// TwinCAT 3 PLC project Execution_Options
// ProgramVersion: 3.1.4023.0
// libraries:
//   Tc2_MC2, * (Beckhoff Automation GmbH)
//   Tc2_Standard, * (Beckhoff Automation GmbH)
//   Tc2_System, * (Beckhoff Automation GmbH)
//   Tc3_Module, * (Beckhoff Automation GmbH)
// project tree:
//   Body Execution/ Body_Task_Base.TcPOU, AxesReset_Body.TcPOU
//   Cycle Method/ AxesReset_Cycle.TcPOU, Cyclic_Task_Base.TcPOU
//   / PlcTask.TcTTO
//   POUs/ MAIN.TcPOU
// real-time tasks:
//   TASK PlcTask: cycle T#10ms, priority 20, ADS port 350

CONFIGURATION Execution_Options
    RESOURCE PLC ON TwinCAT3
        TASK PlcTask(INTERVAL := T#10ms, PRIORITY := 20);
        PROGRAM MAIN WITH PlcTask : MAIN;
    END_RESOURCE
END_CONFIGURATION

// ---- POUs/MAIN.TcPOU
PROGRAM MAIN
VAR
	Axis : AXIS_REF;
	BodyExecution_AxisReset : AxesReset_Body(Axis);
	CycleExecution_AxesReset : AxesReset_Cycle(Axis);
	
END_VAR

///////////////Cycle Call for Body execution//////////////
BodyExecution_AxisReset();


///////////////Cycle Call for Cycle execution////////////
CycleExecution_AxesReset.Cycle();

END_PROGRAM

// ---- Body Execution/AxesReset_Body.TcPOU
FUNCTION_BLOCK AxesReset_Body EXTENDS Body_Task_Base
VAR_INPUT
END_VAR
VAR_OUTPUT
END_VAR
VAR
	resetMover : Tc2_MC2.MC_Reset;
	_axis : REFERENCE TO Tc2_MC2.AXIS_REF;
	_ResetMover : BOOL;
	state : INT;

END_VAR

CASE State OF
	0:
		IF _ResetMover THEN
			_done := FALSE;
			_error := FALSE;
			_busy := TRUE;
			resetMover.Execute := TRUE;
			IF resetMover.Busy THEN
				State := 10;
				_ResetMover := FALSE;
			END_IF
		END_IF
	
	10:
		IF NOT resetMover.Busy THEN
			IF resetMover.Done THEN
				_done := TRUE;
			ELSIF resetMover.Error THEN
				_error := TRUE;
			END_IF
			_busy := FALSE;
			resetMover.Execute := FALSE;
			State := 0;
		END_IF
END_CASE

resetMover(Axis := _axis);

METHOD Abort : BOOL
resetMover.Execute := FALSE;
_busy := FALSE;
_ResetMover := FALSE;
Abort := TRUE;
State := 0;
END_METHOD

PROPERTY Busy : BOOL
GET
Busy := _busy;
END_GET
END_PROPERTY

PROPERTY Done : BOOL
GET
Done := _done;
END_GET
END_PROPERTY

PROPERTY Error : BOOL
GET
Error := _error;
END_GET
END_PROPERTY

METHOD Execute : BOOL
VAR_INPUT
END_VAR
Execute := _ResetMover := true;
END_METHOD

METHOD FB_init : BOOL
VAR_INPUT
	bInitRetains : BOOL; // if TRUE, the retain variables are initialized (warm start / cold start)
	bInCopyCode : BOOL;  // if TRUE, the instance afterwards gets moved into the copy code (online change)
	axis : reference TO AXIS_REF;
END_VAR
_axis REF= axis;
END_METHOD

END_FUNCTION_BLOCK

// ---- Body Execution/Body_Task_Base.TcPOU
FUNCTION_BLOCK ABSTRACT Body_Task_Base
VAR
	_busy : BOOL;
	_error : BOOL;
	_done : BOOL;
END_VAR

METHOD Abort : BOOL
VAR_INPUT
END_VAR
END_METHOD

PROPERTY Busy : bool
GET
Busy := _busy;
END_GET
END_PROPERTY

PROPERTY Done : bool
GET
Done := _done;
END_GET
END_PROPERTY

PROPERTY Error : bool
GET
Error := _error;
END_GET
END_PROPERTY

END_FUNCTION_BLOCK

// ---- Cycle Method/AxesReset_Cycle.TcPOU
FUNCTION_BLOCK AxesReset_Cycle EXTENDS Cyclic_Task_Base
VAR_INPUT
END_VAR
VAR_OUTPUT
END_VAR
VAR
	resetMover : Tc2_MC2.MC_Reset;
	_axis : REFERENCE TO Tc2_MC2.AXIS_REF;
	_ResetMover : BOOL;
	state : INT;
END_VAR

METHOD Abort : BOOL
VAR_INPUT
END_VAR
resetMover.Execute := FALSE;
_busy := FALSE;
_ResetMover := FALSE;
Abort := TRUE;
State := 0;
END_METHOD

METHOD Cycle : BOOL
VAR_INPUT
END_VAR
CASE State OF
	0:
		IF _ResetMover THEN
			_done := FALSE;
			_error := FALSE;
			_busy := TRUE;
			resetMover.Execute := TRUE;
			IF resetMover.Busy THEN
				State := 10;
				_ResetMover := FALSE;
			END_IF
		END_IF
	
	10:
		IF NOT resetMover.Busy THEN
			IF resetMover.Done THEN
				_done := TRUE;
			ELSIF resetMover.Error THEN
				_error := TRUE;
			END_IF
			_busy := FALSE;
			resetMover.Execute := FALSE;
			State := 0;
		END_IF
END_CASE

resetMover(Axis := _axis);
END_METHOD

METHOD Execute : BOOL
VAR_INPUT
END_VAR
Execute := _ResetMover := true;
END_METHOD

METHOD FB_init : BOOL
VAR_INPUT
	bInitRetains : BOOL; // if TRUE, the retain variables are initialized (warm start / cold start)
	bInCopyCode : BOOL;  // if TRUE, the instance afterwards gets moved into the copy code (online change)
	axis : reference TO AXIS_REF;
END_VAR
_axis REF= axis;
END_METHOD

END_FUNCTION_BLOCK

// ---- Cycle Method/Cyclic_Task_Base.TcPOU
FUNCTION_BLOCK PUBLIC ABSTRACT Cyclic_Task_Base
VAR
	_busy : BOOL;
	_error : BOOL;
	_done : BOOL;
END_VAR

METHOD Abort : BOOL
VAR_INPUT
END_VAR
END_METHOD

PROPERTY Busy : bool
GET
Busy := _busy;
END_GET
END_PROPERTY

METHOD Cycle : BOOL
VAR_INPUT
END_VAR
END_METHOD

PROPERTY Done : bool
GET
Done := _done;
END_GET
END_PROPERTY

PROPERTY Error : bool
GET
Error := _error;
END_GET
END_PROPERTY

END_FUNCTION_BLOCK
